FUNCTION_BLOCK FB_WDL
VAR_INPUT
END_VAR
VAR_OUTPUT
END_VAR
VAR (* VAR philipp*)
	System_Blockheizkraftwerk_921				: FB_System_BHKW_921;
	System_Blockheizkraftwerk_922				: FB_System_BHKW_922;
	System_Aussenfassadenaktivierung_600		: FB_System_AFA_600;
	System_Waermetauscher_915					: FB_System_WT_HWW_915;
	System_Absorptionskaeltemaschine_941		: FB_System_AKM_941;
	System_Brennwertkessel_931					: FB_System_BWK_931;
	System_Kaeltekompressor_KW_145				: FB_System_KKKW_145;
	WT_Betrieb: BOOL := FALSE;

	System_Heizstaebe_131_KW					: FB_System_HS_131;
	System_Heizstaebe_231_WW					: FB_System_HS_231;
	Lueftungsklappe_Keller						: FB_SV;
	System_Waermepumpe_946						: FB_System_WP_946;
	Timer1: TOF;
END_VAR
VAR // added by the converter: edge detectors and wires of the graphical bodies
    _w1, _w2, _w3, _w4 : ANY;
END_VAR

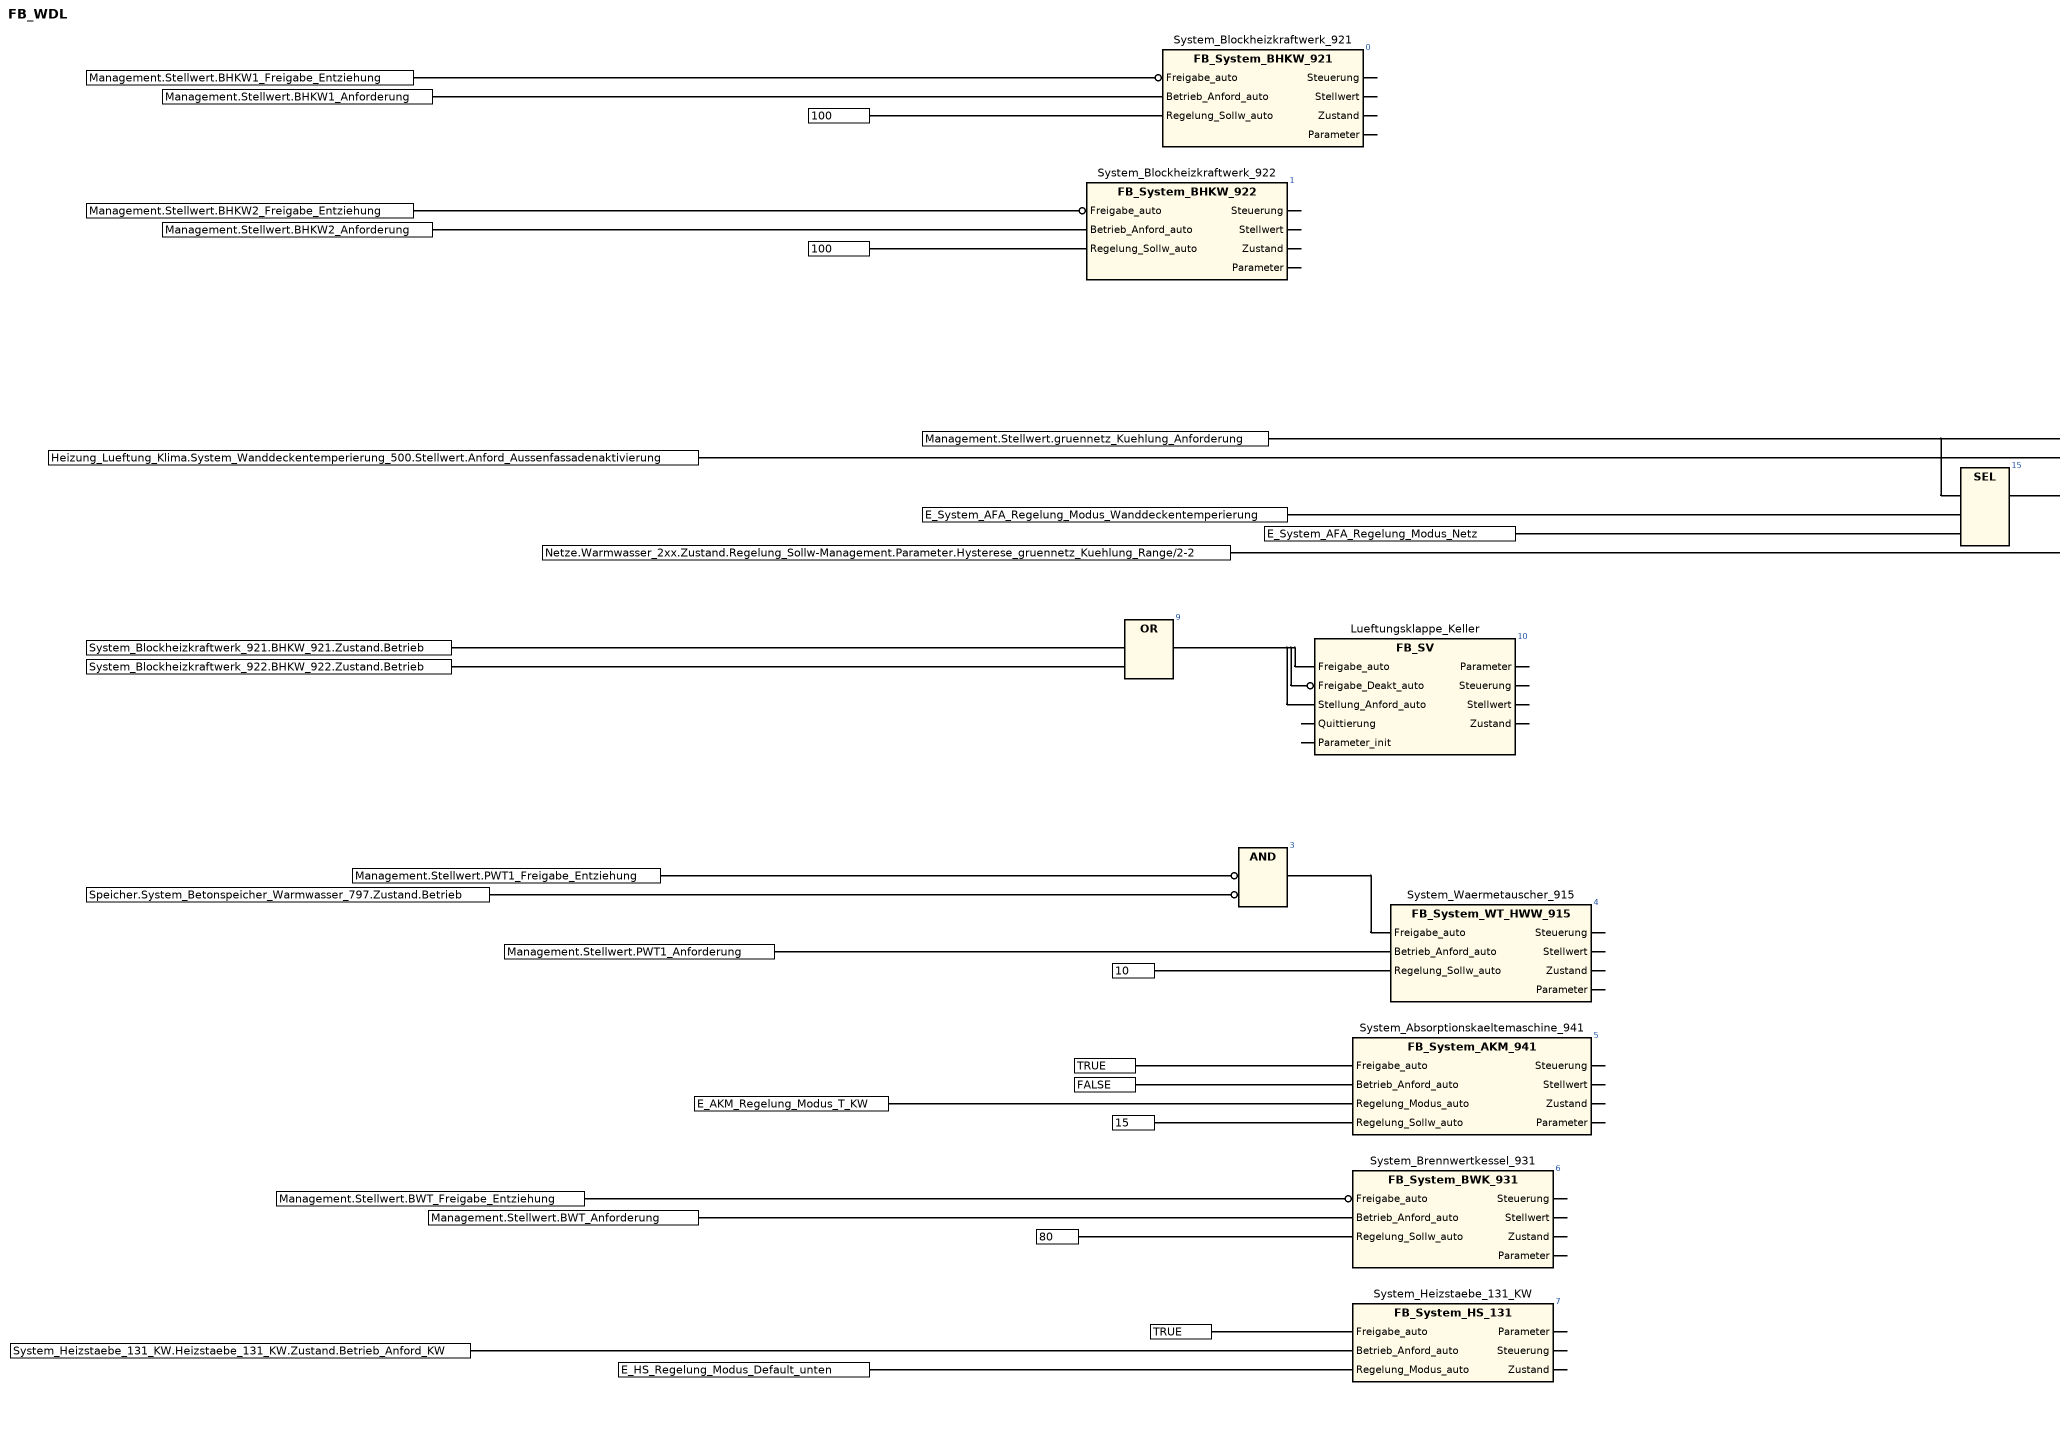
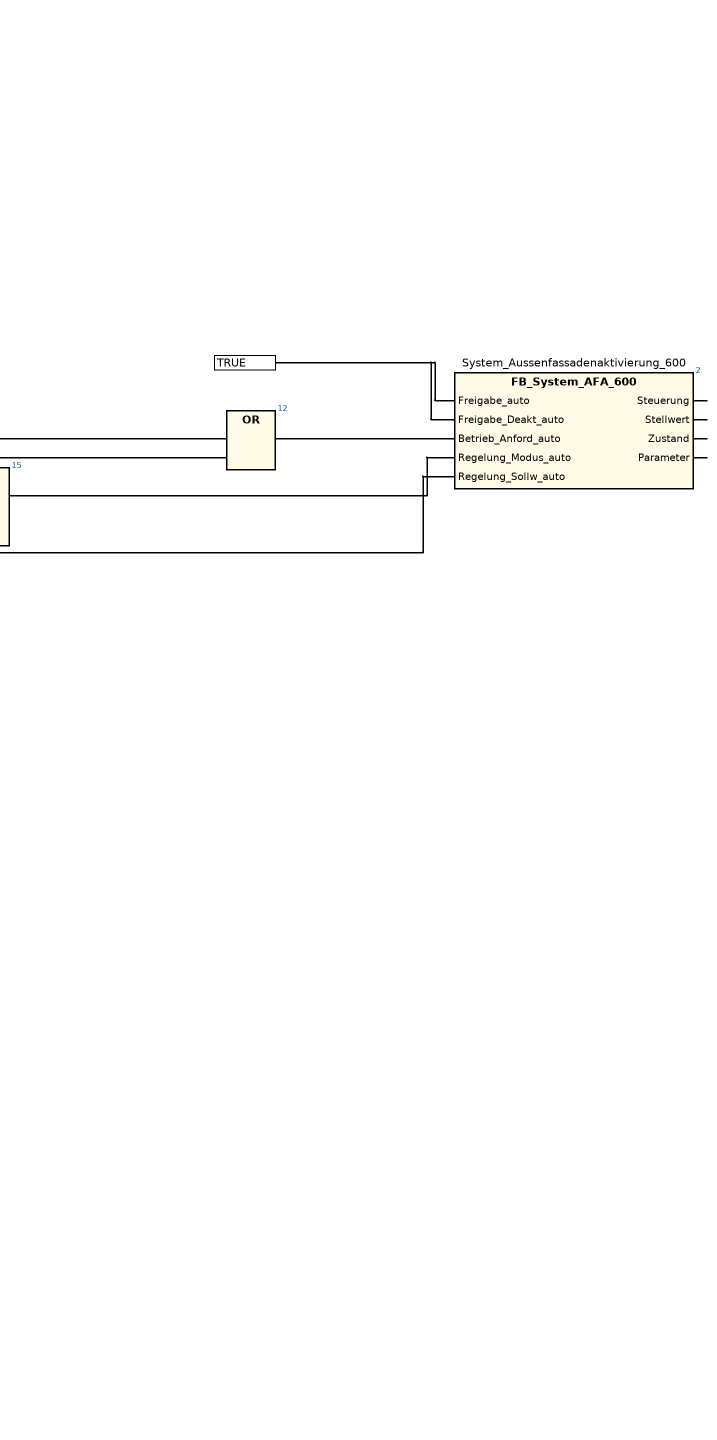
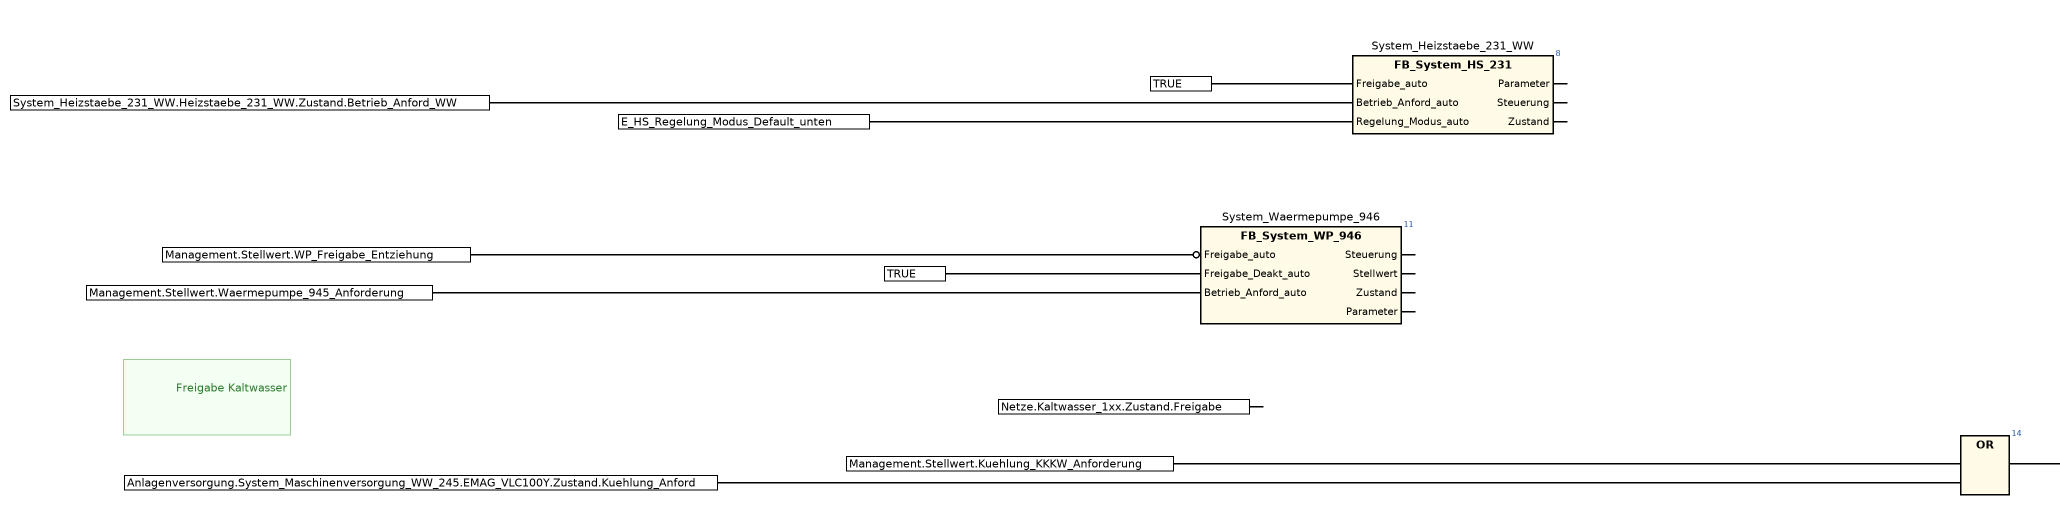
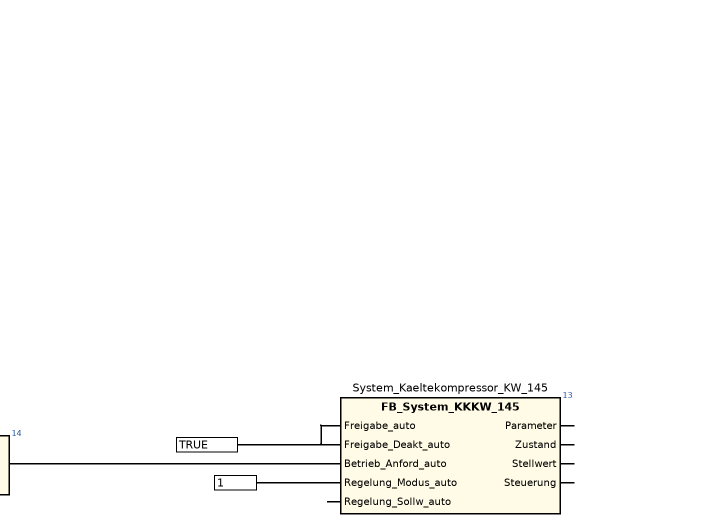
System_Blockheizkraftwerk_921(
    Freigabe_auto := NOT Management.Stellwert.BHKW1_Freigabe_Entziehung,
    Betrieb_Anford_auto := Management.Stellwert.BHKW1_Anforderung,
    Regelung_Sollw_auto := 100); // FB_System_BHKW_921
System_Blockheizkraftwerk_922(
    Freigabe_auto := NOT Management.Stellwert.BHKW2_Freigabe_Entziehung,
    Betrieb_Anford_auto := Management.Stellwert.BHKW2_Anforderung,
    Regelung_Sollw_auto := 100); // FB_System_BHKW_922
System_Aussenfassadenaktivierung_600(
    Freigabe_auto := TRUE,
    Freigabe_Deakt_auto := TRUE,
    Betrieb_Anford_auto := _w1,
    Regelung_Modus_auto := _w2,
    Regelung_Sollw_auto := Netze.Warmwasser_2xx.Zustand.Regelung_Sollw-Management.Parameter.Hysterese_gruennetz_Kuehlung_Range/2-2); // FB_System_AFA_600
System_Waermetauscher_915(
    Freigabe_auto := NOT Management.Stellwert.PWT1_Freigabe_Entziehung AND NOT Speicher.System_Betonspeicher_Warmwasser_797.Zustand.Betrieb,
    Betrieb_Anford_auto := Management.Stellwert.PWT1_Anforderung,
    Regelung_Sollw_auto := 10); // FB_System_WT_HWW_915
System_Absorptionskaeltemaschine_941(
    Freigabe_auto := TRUE,
    Betrieb_Anford_auto := FALSE,
    Regelung_Modus_auto := E_AKM_Regelung_Modus_T_KW,
    Regelung_Sollw_auto := 15); // FB_System_AKM_941
System_Brennwertkessel_931(
    Freigabe_auto := NOT Management.Stellwert.BWT_Freigabe_Entziehung,
    Betrieb_Anford_auto := Management.Stellwert.BWT_Anforderung,
    Regelung_Sollw_auto := 80); // FB_System_BWK_931
System_Heizstaebe_131_KW(
    Freigabe_auto := TRUE,
    Betrieb_Anford_auto := System_Heizstaebe_131_KW.Heizstaebe_131_KW.Zustand.Betrieb_Anford_KW,
    Regelung_Modus_auto := E_HS_Regelung_Modus_Default_unten); // FB_System_HS_131
System_Heizstaebe_231_WW(
    Freigabe_auto := TRUE,
    Betrieb_Anford_auto := System_Heizstaebe_231_WW.Heizstaebe_231_WW.Zustand.Betrieb_Anford_WW,
    Regelung_Modus_auto := E_HS_Regelung_Modus_Default_unten); // FB_System_HS_231
_w3 := System_Blockheizkraftwerk_921.BHKW_921.Zustand.Betrieb OR System_Blockheizkraftwerk_922.BHKW_922.Zustand.Betrieb;
Lueftungsklappe_Keller(Freigabe_auto := _w3, Freigabe_Deakt_auto := NOT _w3, Stellung_Anford_auto := _w3); // FB_SV
System_Waermepumpe_946(
    Freigabe_auto := NOT Management.Stellwert.WP_Freigabe_Entziehung,
    Freigabe_Deakt_auto := TRUE,
    Betrieb_Anford_auto := Management.Stellwert.Waermepumpe_945_Anforderung); // FB_System_WP_946
_w1 := Management.Stellwert.gruennetz_Kuehlung_Anforderung OR Heizung_Lueftung_Klima.System_Wanddeckentemperierung_500.Stellwert.Anford_Aussenfassadenaktivierung;
System_Kaeltekompressor_KW_145(
    Freigabe_auto := TRUE,
    Freigabe_Deakt_auto := TRUE,
    Betrieb_Anford_auto := _w4,
    Regelung_Modus_auto := 1); // FB_System_KKKW_145
// 							Freigabe Kaltwasser
//
//
_w4 := Management.Stellwert.Kuehlung_KKKW_Anforderung OR Anlagenversorgung.System_Maschinenversorgung_WW_245.EMAG_VLC100Y.Zustand.Kuehlung_Anford;
_w2 := SEL(Management.Stellwert.gruennetz_Kuehlung_Anforderung, E_System_AFA_Regelung_Modus_Wanddeckentemperierung, E_System_AFA_Regelung_Modus_Netz);
// Netze.Kaltwasser_1xx.Zustand.Freigabe: input not connected

END_FUNCTION_BLOCK

(* stored: Version 1.1.0.1, ProductVersion 3.1.4024.9
   POU FB_WDL: Id {fb0f0b2a-3883-43ef-ac25-f61ab58a6e43}, SpecialFunc None *)
